TYPE IoStageStruct :
STRUCT
    InputLoadingPosition AT %I* : INT;
    InputProcessPosition AT %I* : INT;	
	
	OutputLoadingPosition AT %Q* : BOOL;
	OutputProcessPosition AT %Q* : BOOL;			
END_STRUCT
END_TYPE

(* stored: Version 1.1.0.1, ProductVersion 3.1.4024.12
   DUT IoStageStruct: Id {4be9c8ab-4b1b-474e-8cab-d89e120b64a9} *)
